ABB RAPID module: TargetDef.mod

MODULE TargetDef
CONST robtarget TOL0_0T1:=[[5.87495484961249, -209.948929822206, 55.199974607377],[0, 0.88684753706352, 0.462062166817809, 0],[-1, 0, -2, 0],[9E9,9E9,9E9,9E9,9E9,9E9]];
CONST robtarget TOL0_1T1:=[[5.62234055193414, -202.858739286579, 35.8261071491754],[0, 0.88684753706352, 0.462062166817809, 0],[-1, 0, -2, 0],[9E9,9E9,9E9,9E9,9E9,9E9]];
CONST robtarget TOL0_1T2:=[[4.98397898868433, -184.941680926626, 25.6156776604893],[0, 0.88684753706352, 0.462062166817809, 0],[-1, 0, -2, 0],[9E9,9E9,9E9,9E9,9E9,9E9]];
CONST robtarget TOL0_2T1:=[[4.89568379013019, -182.463476854714, 25.3040810063602],[0, 0.88684753706352, 0.462062166817809, 0],[-1, 0, -2, 0],[9E9,9E9,9E9,9E9,9E9,9E9]];
CONST robtarget TOL0_2T2:=[[4.80677150236914, -179.967952781144, 25.199974607377],[0, 0.88684753706352, 0.462062166817809, 0],[-1, 0, -2, 0],[9E9,9E9,9E9,9E9,9E9,9E9]];
CONST robtarget TOL0_3T1:=[[4.74728249481166, -178.298524485788, 25.1999746073769],[0, 0.88684753706352, 0.462062166817809, 0],[-1, 0, -2, 0],[9E9,9E9,9E9,9E9,9E9,9E9]];
CONST robtarget TOL0_4T1:=[[4.68786399989119, -176.629093681283, 25.199974607377],[0, 0.88684753706352, 0.462062166817809, 0],[-1, 0, -2, 0],[9E9,9E9,9E9,9E9,9E9,9E9]];
CONST robtarget TOL0_5T1:=[[4.11392451424888, -159.986640927652, 25.199974607377],[0, 0.88684753706352, 0.462062166817809, 0],[-1, 0, -2, 0],[9E9,9E9,9E9,9E9,9E9,9E9]];
CONST robtarget TOL0_6T1:=[[4.16406846873616, -158.042748709129, 25.1999105550075],[0, 0.88684753706352, 0.462062166817809, 0],[-1, 0, -2, 0],[9E9,9E9,9E9,9E9,9E9,9E9]];
CONST robtarget TOL0_7T1:=[[4.21439940943662, -156.098861429512, 25.1997536242781],[0, 0.88684753706352, 0.462062166817809, 0],[-1, 0, -2, 0],[9E9,9E9,9E9,9E9,9E9,9E9]];
CONST robtarget TOL0_8T1:=[[4.26487731018307, -154.154977990189, 25.199556654764],[0, 0.88684753706352, 0.462062166817809, 0],[-1, 1, -2, 0],[9E9,9E9,9E9,9E9,9E9,9E9]];
CONST robtarget TOL0_9T1:=[[4.31546214481006, -152.211097292488, 25.1993724860406],[0, 0.88684753706352, 0.462062166817809, 0],[-1, 1, -2, 0],[9E9,9E9,9E9,9E9,9E9,9E9]];
CONST robtarget TOL0_10T1:=[[4.36611388715329, -150.267218237672, 25.199253957683],[0, 0.88684753706352, 0.462062166817809, 0],[-1, 1, -2, 0],[9E9,9E9,9E9,9E9,9E9,9E9]];
CONST robtarget TOL0_11T1:=[[4.41679251104966, -148.32333972694, 25.1992539092665],[0, 0.88684753706352, 0.462062166817809, 0],[-1, 1, -2, 0],[9E9,9E9,9E9,9E9,9E9,9E9]];
CONST robtarget TOL0_12T1:=[[4.46745799033829, -146.379460661428, 25.1994251803665],[0, 0.88684753706352, 0.462062166817809, 0],[-1, 1, -2, 0],[9E9,9E9,9E9,9E9,9E9,9E9]];
CONST robtarget TOL0_13T1:=[[4.51807029885896, -144.435579942209, 25.1998206105581],[0, 0.88684753706352, 0.462062166817809, 0],[-1, 1, -2, 0],[9E9,9E9,9E9,9E9,9E9,9E9]];
CONST robtarget TOL0_14T1:=[[4.56860145931284, -142.491696832888, 25.2004340400337],[5.78808521166299E-05, -0.886847503502857, -0.462062165385235, -0.000239791711974077],[-1, 1, -2, 0],[9E9,9E9,9E9,9E9,9E9,9E9]];
CONST robtarget TOL0_15T1:=[[4.61907572015895, -140.547812172846, 25.2011438240197],[5.69174071655991E-06, 0.886847487536317, 0.462062177876197, 0.000278557770932622],[-1, 1, -2, 0],[9E9,9E9,9E9,9E9,9E9,9E9]];
CONST robtarget TOL0_16T1:=[[4.66953139612423, -138.603927209032, 25.2017324708743],[9.1999702878942E-05, 0.886847479230205, 0.462062185016766, 0.0002780226918304],[-1, 1, -2, 0],[9E9,9E9,9E9,9E9,9E9,9E9]];
CONST robtarget TOL0_17T1:=[[4.72000680111523, -136.660043190099, 25.2019991082225],[0.000194257642923755, 0.88684748453669, 0.462062172983582, 0.000223008078127303],[-1, 1, -2, 0],[9E9,9E9,9E9,9E9,9E9,9E9]];
CONST robtarget TOL0_18T1:=[[4.77054024868323, -134.716161363558, 25.2017428446979],[0.000305354655708716, 0.886847499341696, 0.462062127896507, 9.8151247610371E-05],[-1, 1, -2, 0],[9E9,9E9,9E9,9E9,9E9,9E9]];
CONST robtarget TOL0_19T1:=[[4.82117005178463, -132.772282975693, 25.2007627603113],[0.00041784330050476, 0.88684749715859, 0.462062040928341, -0.000111909145824577],[-1, 1, -2, 0],[9E9,9E9,9E9,9E9,9E9,9E9]];
CONST robtarget TOL0_20T1:=[[4.87193452255457, -130.828409271538, 25.1988578965212],[0.000523950911211992, 0.886847413047882, 0.462061914798928, -0.000422300923804722],[-1, 1, -2, 0],[9E9,9E9,9E9,9E9,9E9,9E9]];
CONST robtarget TOL0_21T1:=[[4.92287197203422, -128.884541494919, 25.1958272463483],[0.000615615291625375, 0.886847124286926, 0.46206177147994, -0.000847642992470561],[-1, 1, -2, 0],[9E9,9E9,9E9,9E9,9E9,9E9]];
CONST robtarget TOL0_22T1:=[[4.97401555483918, -126.940680952348, 25.1914949656618],[0.000644077831250294, 0.88684637798251, 0.46206172300607, -0.00143218564139338],[-1, 1, -2, 0],[9E9,9E9,9E9,9E9,9E9,9E9]];
CONST robtarget TOL0_23T1:=[[5.02537610710971, -124.996829121411, 25.1858015434017],[0.000673094305604695, 0.886844839539391, 0.462061777689024, -0.00216590056703986],[-1, 1, -2, 0],[9E9,9E9,9E9,9E9,9E9,9E9]];
CONST robtarget TOL0_24T1:=[[5.076958425822, -123.052987547218, 25.1787027683325],[0.000634581591898641, 0.886842136683072, 0.462062165434973, -0.00302938659633397],[-1, 1, -2, 0],[9E9,9E9,9E9,9E9,9E9,9E9]];
CONST robtarget TOL0_25T1:=[[5.12876731366958, -121.109157762365, 25.170161326942],[0.000531980538052365, 0.886837822825442, 0.462063048412129, -0.00401650283548481],[-1, 1, -2, 0],[9E9,9E9,9E9,9E9,9E9,9E9]];
CONST robtarget TOL0_26T1:=[[5.18080757241205, -119.165341299386, 25.1601399052154],[0.000368612428769883, 0.886831406094208, 0.462064598841902, -0.00512130714948808],[-1, 1, -2, 0],[9E9,9E9,9E9,9E9,9E9,9E9]];
CONST robtarget TOL0_27T1:=[[5.23308400297003, -117.221539690753, 25.1486011886477],[0.000147683364606522, 0.886822360123474, 0.462066996155013, -0.00633804693409372],[-1, 1, -2, 0],[9E9,9E9,9E9,9E9,9E9,9E9]];
CONST robtarget TOL0_28T1:=[[5.28560140550417, -115.277754468888, 25.1355078617056],[0.00012771642930868, -0.886810133767952, -0.462070424447913, 0.00766114779298364],[-1, 1, -2, 0],[9E9,9E9,9E9,9E9,9E9,9E9]];
CONST robtarget TOL0_29T1:=[[5.33836457940834, -113.3339871662, 25.1208226029927],[0.000454651248535902, -0.886794159972504, -0.462075070302794, 0.00908518219806045],[-1, 1, -2, 0],[9E9,9E9,9E9,9E9,9E9,9E9]];
CONST robtarget TOL0_30T1:=[[5.39137403539576, -111.390239241959, 25.1045122999512],[0.000830249094422553, -0.886773863455627, -0.462081120469981, 0.0106048990390756],[-1, 1, -2, 0],[9E9,9E9,9E9,9E9,9E9,9E9]];
CONST robtarget TOL0_31T1:=[[5.44461167530778, -109.446511823294, 25.0865606840709],[0.00125172016397042, -0.886748668292076, -0.462088759922859, 0.0122151721975377],[-1, 1, -2, 0],[9E9,9E9,9E9,9E9,9E9,9E9]];
CONST robtarget TOL0_32T1:=[[5.49805438484623, -107.502805944353, 25.0669557018495],[0.00171636213020819, -0.88671800451786, -0.462098170119577, 0.0139109933880112],[-1, 1, -2, 0],[9E9,9E9,9E9,9E9,9E9,9E9]];
CONST robtarget TOL0_33T1:=[[5.5516790497652, -105.559122639288, 25.0456852980213],[0.00222155399052518, -0.88668131405112, -0.462109527403577, 0.0156874693080021],[-1, 1, -2, 0],[9E9,9E9,9E9,9E9,9E9,9E9]];
CONST robtarget TOL0_34T1:=[[5.60546255581983, -103.615462942265, 25.0227374157007],[0.00276475085799574, -0.886638056102518, -0.462123001539547, 0.0175398138964316],[-1, 1, -2, 0],[9E9,9E9,9E9,9E9,9E9,9E9]];
CONST robtarget TOL0_35T1:=[[5.65938178871409, -101.671827887463, 24.9980999965197],[0.00334347917684389, -0.886587712061935, -0.462138754385235, 0.0194633415178935],[-1, 1, -2, 0],[9E9,9E9,9E9,9E9,9E9,9E9]];
CONST robtarget TOL0_36T1:=[[5.71341363405236, -99.7282185090801, 24.9717609807619],[0.0039553323360096, -0.886529789897628, -0.462156938690893, 0.0214534610270855],[-1, 1, -2, 0],[9E9,9E9,9E9,9E9,9E9,9E9]];
CONST robtarget TOL0_37T1:=[[5.76753497738014, -97.7846358413115, 24.9437083094337],[0.0045979493814297, -0.886463827969139, -0.46217769698422, 0.0235056796147047],[-1, 1, -2, 0],[9E9,9E9,9E9,9E9,9E9,9E9]];
CONST robtarget TOL0_38T1:=[[5.82172119826316, -95.8410808542579, 24.9139307673251],[0.00526886801727961, -0.886389397616001, -0.462201160277871, 0.0256156643784414],[-1, 1, -2, 0],[9E9,9E9,9E9,9E9,9E9,9E9]];
CONST robtarget TOL0_39T1:=[[5.87594113313077, -93.8975542480642, 24.8824204552068],[0.0059658038800925, -0.886306109324248, -0.46222744753722, 0.0277790658915003],[-1, 1, -2, 0],[9E9,9E9,9E9,9E9,9E9,9E9]];
CONST robtarget TOL0_40T1:=[[5.93016185341133, -91.9540566517558, 24.8491703063232],[0.00668656550503767, -0.886213614964218, -0.462256664707816, 0.0299915725997466],[-1, 1, -2, 0],[9E9,9E9,9E9,9E9,9E9,9E9]];
CONST robtarget TOL0_41T1:=[[5.98435043019924, -90.0105886943894, 24.8141732528904],[0.00742900624154073, -0.886111609894809, -0.462288903935541, 0.0322489375634248],[-1, 1, -2, 0],[9E9,9E9,9E9,9E9,9E9,9E9]];
CONST robtarget TOL0_42T1:=[[6.03847393420563, -88.0671510050547, 24.7774222262555],[0.00819102143652073, -0.885999835193581, -0.462324242939227, 0.0345469766469368],[-1, 1, -2, 0],[9E9,9E9,9E9,9E9,9E9,9E9]];
CONST robtarget TOL0_43T1:=[[6.09249943571575, -86.1237442128753, 24.7389101570525],[0.00897054595159374, -0.885878079539174, -0.462362744481674, 0.036881567383844],[-1, 1, -2, 0],[9E9,9E9,9E9,9E9,9E9,9E9]];
CONST robtarget TOL0_44T1:=[[6.14639400455496, -84.1803689470091, 24.6986299753559],[0.00976555199443826, -0.885746180751911, -0.462404455938409, 0.0392486484601787],[-1, 1, -2, 0],[9E9,9E9,9E9,9E9,9E9,9E9]];
CONST robtarget TOL0_45T1:=[[6.2001247100614, -82.2370258366481, 24.656574610829],[0.0105740472453268, -0.885604026997849, -0.462449408963551, 0.0416442197586716],[-1, 1, -2, 0],[9E9,9E9,9E9,9E9,9E9,9E9]];
CONST robtarget TOL0_46T1:=[[6.2536573860541, -80.2937157169943, 24.6127341371022],[0.0113941391592412, -0.885451558975314, -0.462497619103059, 0.0440643010271058],[-1, 1, -2, 0],[9E9,9E9,9E9,9E9,9E9,9E9]];
CONST robtarget TOL0_47T1:=[[6.30695259345345, -78.3504402383671, 24.5670871945443],[0.0122245639579626, -0.885288779804087, -0.462549084720571, 0.0465046300188573],[-1, 1, -2, 0],[9E9,9E9,9E9,9E9,9E9,9E9]];
CONST robtarget TOL0_48T1:=[[6.35996949801029, -76.4072012510752, 24.5196096457906],[0.0130635804060093, -0.885115740486263, -0.462603787181224, 0.0489612591343337],[-1, 1, -2, 0],[9E9,9E9,9E9,9E9,9E9,9E9]];
CONST robtarget TOL0_49T1:=[[6.41266726646654, -74.4640006050592, 24.4702773733228],[0.0139093019982725, -0.884932542700248, -0.462661691416617, 0.0514303945494261],[-1, 1, -2, 0],[9E9,9E9,9E9,9E9,9E9,9E9]];
CONST robtarget TOL0_50T1:=[[6.46500506498899, -72.520840150277, 24.4190662601734],[0.0147598699942932, -0.884739340551065, -0.462722746086731, 0.0539083089418833],[-1, 1, -2, 0],[9E9,9E9,9E9,9E9,9E9,9E9]];
CONST robtarget TOL0_51T1:=[[6.51694205924105, -70.5777217367015, 24.3659521900665],[0.0156134533099272, -0.884536339837173, -0.462786883826999, 0.0563913445565212],[-1, 1, -2, 0],[9E9,9E9,9E9,9E9,9E9,9E9]];
CONST robtarget TOL0_52T1:=[[6.56843741446033, -68.634647214319, 24.3109110475456],[0.0164682485958798, -0.884323797009536, -0.462854021586783, 0.0588759163984978],[-1, 1, -2, 0],[9E9,9E9,9E9,9E9,9E9,9E9]];
CONST robtarget TOL0_53T1:=[[6.61945029554181, -66.6916184331267, 24.25391871809],[0.0173224804765711, -0.884102017837447, -0.462924061054783, 0.0613585154843354],[-1, 1, -2, 0],[9E9,9E9,9E9,9E9,9E9,9E9]];
CONST robtarget TOL0_54T1:=[[6.66994435104448, -64.7486365163287, 24.1949689968205],[0.0181744089212188, -0.883871354009737, -0.462996889732181, 0.063835730744511],[-1, 1, -2, 0],[9E9,9E9,9E9,9E9,9E9,9E9]];
CONST robtarget TOL0_55T1:=[[6.7199019031716, -62.805699700113, 24.1341272804838],[0.0190218342643242, -0.883632185515794, -0.463072384977798, 0.066304576107361],[-1, 1, -2, 0],[9E9,9E9,9E9,9E9,9E9,9E9]];
CONST robtarget TOL0_56T1:=[[6.76931020604997, -60.8628054877942, 24.0714774096135],[0.0198573737794578, -0.883384829109368, -0.463150429844447, 0.0687648728705193],[-1, 0, -2, 0],[9E9,9E9,9E9,9E9,9E9,9E9]];
CONST robtarget TOL0_57T1:=[[6.81815645803619, -58.9199513943938, 24.0071027577105],[0.0206778301201626, -0.883129717086152, -0.46323088464036, 0.0712143079455536],[-1, 0, -2, 0],[9E9,9E9,9E9,9E9,9E9,9E9]];
CONST robtarget TOL0_58T1:=[[6.86642783302506, -56.9771349397499, 23.9410865196908],[0.0214816257464342, -0.882867352992543, -0.463313591712299, 0.0736497964008017],[-1, 0, -2, 0],[9E9,9E9,9E9,9E9,9E9,9E9]];
CONST robtarget TOL0_59T1:=[[6.91411150360364, -55.0343536436539, 23.8735118903307],[0.0222672059395263, -0.882598279750095, -0.46339838054372, 0.0760683181835714],[-1, 0, -2, 0],[9E9,9E9,9E9,9E9,9E9,9E9]];
CONST robtarget TOL0_60T1:=[[6.96119441598756, -53.0916050709859, 23.8044606758834],[0.023045541467769, -0.882323362092062, -0.463485011503932, 0.0784603838648393],[-1, 0, -2, 0],[9E9,9E9,9E9,9E9,9E9,9E9]];
CONST robtarget TOL0_61T1:=[[7.00766329729066, -51.1488868294857, 23.7340135480734],[0.0238379753498431, -0.882043756945659, -0.463573176999837, 0.0808113316972624],[-1, 0, -2, 0],[9E9,9E9,9E9,9E9,9E9,9E9]];
CONST robtarget TOL0_62T1:=[[7.05348992599602, -49.2062003980425, 23.6621651291686],[0.0246434226405345, -0.881760150918272, -0.463662654617083, 0.0831184737984602],[-1, 0, -2, 0],[9E9,9E9,9E9,9E9,9E9,9E9]];
CONST robtarget TOL0_63T1:=[[7.09858462534561, -47.2635630423646, 23.5885558995094],[0.0254603521153771, -0.881473231922942, -0.463753217597252, 0.0853795352627361],[-1, 0, -2, 0],[9E9,9E9,9E9,9E9,9E9,9E9]];
CONST robtarget TOL0_64T1:=[[7.14284253298126, -45.3209959322502, 23.5127389692874],[0.0262767684505692, -0.881183417162999, -0.46384470052432, 0.0875980054124462],[-1, 0, -2, 0],[9E9,9E9,9E9,9E9,9E9,9E9]];
CONST robtarget TOL0_65T1:=[[7.18616220901009, -43.3785195720567, 23.4342856300351],[0.0269162483623758, -0.880886836321344, -0.463937962561879, 0.0898635858610179],[-1, 0, -2, 0],[9E9,9E9,9E9,9E9,9E9,9E9]];
CONST robtarget TOL0_66T1:=[[7.22844016516217, -41.4361548561847, 23.3527545172302],[0.0273156512506206, -0.880582353172387, -0.464033139854085, 0.0922053121858804],[-1, 0, -2, 0],[9E9,9E9,9E9,9E9,9E9,9E9]];
CONST robtarget TOL0_67T1:=[[7.26957169093038, -39.493922882487, 23.2676974031319],[0.0274736194950504, -0.880270370217772, -0.464129743785235, 0.0946195354161044],[-1, 0, -2, 0],[9E9,9E9,9E9,9E9,9E9,9E9]];
CONST robtarget TOL0_68T1:=[[7.30945207826227, -37.5518447104956, 23.1786661163437],[0.0273882713081452, -0.879951240672993, -0.464227015451949, 0.0971029080789399],[-1, 0, -2, 0],[9E9,9E9,9E9,9E9,9E9,9E9]];
CONST robtarget TOL0_69T1:=[[7.34797711476068, -35.6099412503439, 23.0852149483144],[0.0270353507422883, -0.87962460427133, -0.464323980346725, 0.0996638683060276],[-1, 0, -2, 0],[9E9,9E9,9E9,9E9,9E9,9E9]];
CONST robtarget TOL0_70T1:=[[7.43410920658374, -35.2152949167019, 23.049134476302],[0.027387152036867, -0.879402536820145, -0.464393137984042, 0.101193554789508],[-1, 0, -2, 0],[9E9,9E9,9E9,9E9,9E9,9E9]];
CONST robtarget TOL0_71T1:=[[7.83197636578603, -33.6097358151834, 22.8847547435323],[0.0287458481344975, -0.878443440770914, -0.464690940547519, 0.107578470683722],[-1, 0, -2, 0],[9E9,9E9,9E9,9E9,9E9,9E9]];
CONST robtarget TOL0_72T1:=[[8.22945422240645, -32.0052187325015, 22.7096518119473],[0.0299679675605213, -0.877402453198319, -0.465012407313013, 0.114150414308576],[-1, 0, -2, 0],[9E9,9E9,9E9,9E9,9E9,9E9]];
CONST robtarget TOL0_73T1:=[[8.62647919807819, -30.4019739957621, 22.522482668734],[0.0310535472491881, -0.876276641963512, -0.465357816872208, 0.120900894241218],[-1, 0, -2, 0],[9E9,9E9,9E9,9E9,9E9,9E9]];
CONST robtarget TOL0_74T1:=[[9.02298779202067, -28.8002318707254, 22.3219045770051],[0.0320062367781418, -0.875061742490296, -0.465727744933963, 0.127828851343795],[-1, 0, -2, 0],[9E9,9E9,9E9,9E9,9E9,9E9]];
CONST robtarget TOL0_75T1:=[[9.41891881577311, -27.2002263124348, 22.106689574242],[0.0328307845960863, -0.873754414135797, -0.466122396477093, 0.134926924160703],[-1, 0, -2, 0],[9E9,9E9,9E9,9E9,9E9,9E9]];
CONST robtarget TOL0_76T1:=[[9.81421180453196, -25.6022037193409, 21.8760718212889],[0.0335410415525868, -0.872351878470698, -0.46654187882036, 0.142182537489597],[-1, 0, -2, 0],[9E9,9E9,9E9,9E9,9E9,9E9]];
CONST robtarget TOL0_77T1:=[[10.2088046734556, -24.0064128875366, 21.6294029478869],[0.0341394073310869, -0.870851111778797, -0.466986180215052, 0.149588600731706],[-1, 0, -2, 0],[9E9,9E9,9E9,9E9,9E9,9E9]];
CONST robtarget TOL0_78T1:=[[10.6026353833184, -22.4131025747239, 21.3660347119904],[0.0346270923135725, -0.869249101594861, -0.467455194957132, 0.15713880667112],[-1, 0, -2, 0],[9E9,9E9,9E9,9E9,9E9,9E9]];
CONST robtarget TOL0_79T1:=[[10.9956381087109, -20.8225410290283, 21.0852936408323],[0.0350053180038412, -0.86754286815456, -0.467948737621279, 0.16482711726006],[-1, 0, -2, 0],[9E9,9E9,9E9,9E9,9E9,9E9]];
CONST robtarget TOL0_80T1:=[[11.387735033502, -19.2350755024655, 20.7864043718172],[0.035275549555721, -0.865729392921139, -0.468466575321836, 0.172647970281056],[-1, 0, -2, 0],[9E9,9E9,9E9,9E9,9E9,9E9]];
CONST robtarget TOL0_81T1:=[[11.7788461517508, -17.6510732111494, 20.4685658049336],[0.0354395435717827, -0.863805699488511, -0.469008415288741, 0.180595843448654],[-1, 0, -2, 0],[9E9,9E9,9E9,9E9,9E9,9E9]];
CONST robtarget TOL0_82T1:=[[12.1688914672051, -16.0709013399982, 20.1309767973821],[0.035499089128212, -0.861768975535691, -0.469573873144648, 0.188664848700458],[-1, 0, -1, 0],[9E9,9E9,9E9,9E9,9E9,9E9]];
CONST robtarget TOL0_83T1:=[[12.5577737734797, -14.4949397020433, 19.7728616566787],[0.0354496734894093, -0.859619255222402, -0.470161502354852, 0.196840591351999],[-1, 0, -1, 0],[9E9,9E9,9E9,9E9,9E9,9E9]];
CONST robtarget TOL0_84T1:=[[12.9453200975713, -12.9236163390144, 19.3935496981315],[0.0352839590064922, -0.857358264143806, -0.470769168972642, 0.205105433097117],[-1, 0, -1, 0],[9E9,9E9,9E9,9E9,9E9,9E9]];
CONST robtarget TOL0_85T1:=[[13.3313368681544, -11.3573707185873, 18.9923973991323],[0.0350023271936787, -0.854984460453189, -0.471395831043085, 0.21345346085223],[-1, 0, -1, 0],[9E9,9E9,9E9,9E9,9E9,9E9]];
CONST robtarget TOL0_86T1:=[[13.715630356576, -9.79664234621814, 18.5687608492739],[0.0346091194395503, -0.852496634607658, -0.472040505657559, 0.221877123320074],[-1, 0, -1, 0],[9E9,9E9,9E9,9E9,9E9,9E9]];
CONST robtarget TOL0_87T1:=[[14.0980062151705, -8.24188693555804, 18.1219996102562],[0.0341140537110323, -0.849894694300878, -0.472702239067701, 0.2303645656758],[-1, 0, -1, 0],[9E9,9E9,9E9,9E9,9E9,9E9]];
CONST robtarget TOL0_88T1:=[[14.4782703339407, -6.6936249152833, 17.6514899462765],[0.0335188844077826, -0.847178241537506, -0.473379814829405, 0.238908062579636],[-1, 0, -1, 0],[9E9,9E9,9E9,9E9,9E9,9E9]];
CONST robtarget TOL0_89T1:=[[14.856319392745, -5.15244264550846, 17.1565742612497],[0.0328272708903672, -0.844345818016324, -0.474072416101428, 0.247503240738359],[-1, 0, -1, 0],[9E9,9E9,9E9,9E9,9E9,9E9]];
CONST robtarget TOL0_90T1:=[[15.2324495482948, -3.61913923974505, 16.6364277633281],[0.0320431726758495, -0.841395948739511, -0.474779283629122, 0.256145904449442],[-1, 0, -1, 0],[9E9,9E9,9E9,9E9,9E9,9E9]];
CONST robtarget TOL0_91T1:=[[15.6067133899127, -2.09441147356056, 16.0903883343992],[0.0311744453603097, -0.838325138427612, -0.475500514305436, 0.264836510194628],[-1, 0, -1, 0],[9E9,9E9,9E9,9E9,9E9,9E9]];
CONST robtarget TOL0_92T1:=[[15.9776026533308, -0.578260587893794, 15.5186930171285],[0.0302074534032609, -0.835141339137625, -0.476231675882653, 0.273550441981555],[-1, 0, -1, 0],[9E9,9E9,9E9,9E9,9E9,9E9]];
CONST robtarget TOL0_93T1:=[[16.3460386010615, 0.928181059726583, 14.9203842450379],[0.0291600686936652, -0.831836088634164, -0.476974944471034, 0.282300043192435],[-1, 0, -1, 0],[9E9,9E9,9E9,9E9,9E9,9E9]];
CONST robtarget TOL0_94T1:=[[16.7116757500925, 2.42427889302336, 14.2949178617212],[0.0280320714161996, -0.82841040669241, -0.477728767810928, 0.291076665951922],[-1, 0, -1, 0],[9E9,9E9,9E9,9E9,9E9,9E9]];
CONST robtarget TOL0_95T1:=[[17.0151361682334, 3.93476049963918, 13.6717584136658],[0.0260567021781286, -0.825274850857875, -0.478314666391687, 0.299094548141088],[-1, 0, -1, 0],[9E9,9E9,9E9,9E9,9E9,9E9]];
CONST robtarget TOL0_96T1:=[[17.1885483413104, 5.48153915463342, 13.0889076997537],[0.0218239495227135, -0.822800320403308, -0.478477261399255, 0.305913154825538],[-1, 0, -1, 0],[9E9,9E9,9E9,9E9,9E9,9E9]];
CONST robtarget TOL0_97T1:=[[17.2254385337467, 7.05325549652198, 12.5497391180146],[0.0144872412219819, -0.821000352955872, -0.478058340683713, 0.311783199019517],[-1, 0, -1, 0],[9E9,9E9,9E9,9E9,9E9,9E9]];
CONST robtarget TOL0_98T1:=[[17.1252319861591, 8.63730799664661, 12.0573412841479],[0.00524659813226371, -0.820201874224259, -0.477043854613766, 0.315706381788983],[-1, 0, -1, 0],[9E9,9E9,9E9,9E9,9E9,9E9]];
CONST robtarget TOL0_99T1:=[[16.8838655266047, 10.2220927847176, 11.6171916385159],[0.00597316665179748, 0.820436524121733, 0.475359131296763, -0.317619154743517],[-1, 0, -1, 0],[9E9,9E9,9E9,9E9,9E9,9E9]];
CONST robtarget TOL0_100T1:=[[16.496459258559, 11.7913593023744, 11.2323677652838],[0.019225135650213, 0.821720532595913, 0.472929037796034, -0.317401773276139],[-1, 0, -1, 0],[9E9,9E9,9E9,9E9,9E9,9E9]];
CONST robtarget TOL0_101T1:=[[15.9620388422879, 13.3292864997246, 10.9035216337546],[0.0343858161198326, 0.823952858276942, 0.469729414294668, -0.315077102204235],[0, 0, -1, 0],[9E9,9E9,9E9,9E9,9E9,9E9]];
CONST robtarget TOL0_102T1:=[[15.2975665242909, 14.8265997654873, 10.6230056722904],[0.0513144276670698, 0.827031767548874, 0.465745710339988, -0.310590112975424],[0, 0, -1, 0],[9E9,9E9,9E9,9E9,9E9,9E9]];
CONST robtarget TOL0_103T1:=[[14.967367080232, 15.4539259643929, 10.5171328666547],[0.0590775300410213, 0.828573423219684, 0.463798553078389, -0.30800459402525],[0, 0, -1, 0],[9E9,9E9,9E9,9E9,9E9,9E9]];
CONST robtarget TOL0_104T1:=[[13.8242741167196, 17.2551838840315, 10.2499142060585],[0.0836930125687464, 0.833774679307542, 0.457206753692931, -0.297955110998864],[0, 0, -1, 0],[9E9,9E9,9E9,9E9,9E9,9E9]];
CONST robtarget TOL0_105T1:=[[12.4848081223101, 18.9224226369913, 10.0402609053551],[0.109534625655401, 0.839498617006178, 0.449720616805198, -0.284597267463337],[0, 0, -1, 0],[9E9,9E9,9E9,9E9,9E9,9E9]];
CONST robtarget TOL0_106T1:=[[10.9536580099233, 20.4227808614128, 9.88079634359366],[0.135438074203304, 0.845217264609808, 0.441778026830691, -0.268507874505003],[0, 0, -1, 0],[9E9,9E9,9E9,9E9,9E9,9E9]];
CONST robtarget TOL0_107T1:=[[9.25279902191795, 21.733940718676, 9.76141824500081],[0.160711130131284, 0.850682329933611, 0.433745809055314, -0.249752035662573],[0, 0, -1, 0],[9E9,9E9,9E9,9E9,9E9,9E9]];
CONST robtarget TOL0_108T1:=[[7.40886096224591, 22.8377253427806, 9.67235716029097],[0.184787474070288, 0.855676877550213, 0.426005724317412, -0.228450855768669],[0, 0, -1, 0],[9E9,9E9,9E9,9E9,9E9,9E9]];
CONST robtarget TOL0_109T1:=[[5.44903033150683, 23.7213019041005, 9.60859755233264],[0.20715683426475, 0.860015923003412, 0.418948401521263, -0.204794763265019],[0, 0, -2, 0],[9E9,9E9,9E9,9E9,9E9,9E9]];
CONST robtarget TOL0_110T1:=[[3.40063086296732, 24.3731686868072, 9.56625582451045],[0.227129911032962, 0.863476298086857, 0.412995568241102, -0.179597735981233],[0, 0, -2, 0],[9E9,9E9,9E9,9E9,9E9,9E9]];
CONST robtarget TOL0_111T1:=[[1.29099086049644, 24.7818685137185, 9.54151159931365],[0.244587840350064, 0.866034249185732, 0.408359653076031, -0.152983206038509],[0, 0, -2, 0],[9E9,9E9,9E9,9E9,9E9,9E9]];
CONST robtarget TOL0_112T1:=[[-0.852267278068496, 24.9384128294188, 9.53145844273632],[0.259577705187279, 0.86767136716036, 0.405165412304917, -0.124927187799793],[0, 0, -2, 0],[9E9,9E9,9E9,9E9,9E9,9E9]];
CONST robtarget TOL0_113T1:=[[-3.00023476448621, 24.844012774621, 9.53644373163792],[0.271889307282029, 0.868342688426414, 0.403531423738877, -0.0960185924566771],[0, 0, -2, 0],[9E9,9E9,9E9,9E9,9E9,9E9]];
CONST robtarget TOL0_114T1:=[[-5.12366624708858, 24.502525867907, 9.55754302843019],[0.28135861594483, 0.868077486512614, 0.403439060009092, -0.0671991927223259],[0, 1, -2, 0],[9E9,9E9,9E9,9E9,9E9,9E9]];
CONST robtarget TOL0_115T1:=[[-7.19333271253106, 23.9178635833248, 9.59591180590405],[0.288314290128393, 0.866942341188987, 0.404733532419318, -0.0384267471548012],[0, 1, -2, 0],[9E9,9E9,9E9,9E9,9E9,9E9]];
CONST robtarget TOL0_116T1:=[[-9.17986849060492, 23.0950990283751, 9.65350899172734],[0.293085784728034, 0.864964080104485, 0.407240030693865, -0.00966541876041895],[0, 1, -2, 0],[9E9,9E9,9E9,9E9,9E9,9E9]];
CONST robtarget TOL0_117T1:=[[-11.0533207749818, 22.0440582483403, 9.73539475274919],[0.295695307915798, 0.862263102822051, 0.410766595359259, 0.0183692821098943],[0, 1, -2, 0],[9E9,9E9,9E9,9E9,9E9,9E9]];
CONST robtarget TOL0_118T1:=[[-12.7872263020506, 20.7794803940538, 9.84738095575494],[0.2964167184953, 0.858955230763517, 0.415060996665293, 0.0453586770936465],[0, 1, -2, 0],[9E9,9E9,9E9,9E9,9E9,9E9]];
CONST robtarget TOL0_119T1:=[[-14.3702073274265, 19.3317230411206, 9.99434809074609],[0.295555093865856, 0.855144094965721, 0.419892824553204, 0.0711742876601827],[0, 1, -2, 0],[9E9,9E9,9E9,9E9,9E9,9E9]];
CONST robtarget TOL0_120T1:=[[-14.8501607304607, 18.8164149185304, 10.0523405697373],[0.294965135682195, 0.853808338616108, 0.421558451563138, 0.0793433145090054],[0, 1, -2, 0],[9E9,9E9,9E9,9E9,9E9,9E9]];
CONST robtarget TOL0_121T1:=[[-16.2076741090664, 17.091805662966, 10.2716810818974],[0.292265376866975, 0.849475896643786, 0.426882422621381, 0.103648674680103],[0, 1, -2, 0],[9E9,9E9,9E9,9E9,9E9,9E9]];
CONST robtarget TOL0_122T1:=[[-17.3579077901645, 15.2330082223245, 10.5535971346291],[0.288191314532163, 0.845270097479071, 0.432176877743502, 0.125249251015019],[0, 1, -2, 0],[9E9,9E9,9E9,9E9,9E9,9E9]];
CONST robtarget TOL0_123T1:=[[-18.2679853277614, 13.2576263755874, 10.9164700516849],[0.282757246693219, 0.841580157683036, 0.437231498642144, 0.143595940861194],[-1, 1, -2, 0],[9E9,9E9,9E9,9E9,9E9,9E9]];
CONST robtarget TOL0_124T1:=[[-18.9282987581193, 11.2022331861768, 11.3709652323788],[0.275865633923922, 0.838802145713515, 0.441892833132222, 0.158239806599144],[-1, 1, -2, 0],[9E9,9E9,9E9,9E9,9E9,9E9]];
CONST robtarget TOL0_125T1:=[[-19.3366998057772, 9.10642946980709, 11.9227671757553],[0.267431534272727, 0.837226195476365, 0.446064871239216, 0.168993499079251],[-1, 1, -2, 0],[9E9,9E9,9E9,9E9,9E9,9E9]];
CONST robtarget TOL0_126T1:=[[-19.4965991647885, 7.00248777750436, 12.5659733328788],[0.257354967513303, 0.837025344316078, 0.449706252013001, 0.175844478358571],[-1, 1, -2, 0],[9E9,9E9,9E9,9E9,9E9,9E9]];
CONST robtarget TOL0_127T1:=[[-19.410921819497, 4.92186687191422, 13.2933999260707],[0.245839935005472, 0.8382198120052, 0.452739413887211, 0.178821967978035],[-1, 1, -2, 0],[9E9,9E9,9E9,9E9,9E9,9E9]];
CONST robtarget TOL0_128T1:=[[-19.0875426396446, 2.89348719239379, 14.097068940899],[0.235289232001358, 0.840599152710681, 0.454569819926168, 0.177195712641664],[-1, 1, -2, 0],[9E9,9E9,9E9,9E9,9E9,9E9]];
CONST robtarget TOL0_129T1:=[[-18.6102716309398, 0.906360223588791, 14.9291384799526],[0.223990247526092, 0.843722572428624, 0.456019413741289, 0.173224952240367],[-1, 1, -2, 0],[9E9,9E9,9E9,9E9,9E9,9E9]];
CONST robtarget TOL0_130T1:=[[-18.1201101074537, -1.09543148925224, 15.7172539691776],[0.21282322284174, 0.84676945109027, 0.457299572124969, 0.169011460717484],[-1, 1, -2, 0],[9E9,9E9,9E9,9E9,9E9,9E9]];
CONST robtarget TOL0_131T1:=[[-17.6268326464086, -3.11441539133411, 16.4581743933638],[0.20183330684969, 0.849710254539164, 0.458425216266941, 0.16462721727502],[-1, 1, -2, 0],[9E9,9E9,9E9,9E9,9E9,9E9]];
CONST robtarget TOL0_132T1:=[[-17.1270050146111, -5.14744898116223, 17.1548989732062],[0.19101493583257, 0.852557577273439, 0.459401526056578, 0.160028464903621],[-1, 1, -2, 0],[9E9,9E9,9E9,9E9,9E9,9E9]];
CONST robtarget TOL0_133T1:=[[-16.6241928732059, -7.19455251544644, 17.806847571344],[0.180407967373584, 0.855290530421207, 0.46024159112668, 0.155269931658141],[-1, 1, -2, 0],[9E9,9E9,9E9,9E9,9E9,9E9]];
CONST robtarget TOL0_134T1:=[[-16.1183745316094, -9.25418664761038, 18.4157406825447],[0.170018618749308, 0.857913209728371, 0.460953206051751, 0.150335410608257],[-1, 1, -2, 0],[9E9,9E9,9E9,9E9,9E9,9E9]];
CONST robtarget TOL0_135T1:=[[-15.6088409760248, -11.3245573025151, 18.9837212306742],[0.159864590327202, 0.860422186707043, 0.461545945455, 0.145231930427976],[-1, 1, -2, 0],[9E9,9E9,9E9,9E9,9E9,9E9]];
CONST robtarget TOL0_136T1:=[[-15.0960787303775, -13.4045453337182, 19.5121722473094],[0.149975300978849, 0.862815177086043, 0.462027176845585, 0.139958090664247],[-1, 1, -2, 0],[9E9,9E9,9E9,9E9,9E9,9E9]];
CONST robtarget TOL0_137T1:=[[-14.5808088220936, -15.493214306599, 20.0023703822673],[0.140372435895946, 0.865088826427405, 0.462406934533967, 0.134524081583902],[-1, 1, -2, 0],[9E9,9E9,9E9,9E9,9E9,9E9]];
CONST robtarget TOL0_138T1:=[[-14.0633726764923, -17.5896421566149, 20.4559695966065],[0.131074018363047, 0.867238384223207, 0.462696844175012, 0.128952770542435],[-1, 1, -2, 0],[9E9,9E9,9E9,9E9,9E9,9E9]];
CONST robtarget TOL0_139T1:=[[-13.5440096366595, -19.6929081775059, 20.8747204007841],[0.122103216966882, 0.869257873169228, 0.462908531594784, 0.12327710945837],[-1, 1, -2, 0],[9E9,9E9,9E9,9E9,9E9,9E9]];
CONST robtarget TOL0_140T1:=[[-13.0229591655849, -21.802091701674, 21.2603737525102],[0.113473998074668, 0.871147612677842, 0.463051803724335, 0.117509641112072],[-1, 1, -2, 0],[9E9,9E9,9E9,9E9,9E9,9E9]];
CONST robtarget TOL0_141T1:=[[-12.5004429779489, -23.9163253349126, 21.6147044837566],[0.105197548023017, 0.872909258683923, 0.463135958174091, 0.111660137202116],[-1, 1, -2, 0],[9E9,9E9,9E9,9E9,9E9,9E9]];
CONST robtarget TOL0_142T1:=[[-11.9766094698917, -26.0349538826794, 21.9395828092331],[0.0972844348343415, 0.8745449114134, 0.463169841914148, 0.105738518058062],[-1, 1, -2, 0],[9E9,9E9,9E9,9E9,9E9,9E9]];
CONST robtarget TOL0_143T1:=[[-11.4515880913778, -28.1573751184934, 22.2369029041797],[0.0897456004067372, 0.876056983401301, 0.463161765321256, 0.0997550409049293],[-1, 1, -2, 0],[9E9,9E9,9E9,9E9,9E9,9E9]];
CONST robtarget TOL0_144T1:=[[-10.9255078273131, -30.2829870216002, 22.5085572693407],[0.082607647437601, 0.877448336990899, 0.463118159041064, 0.0937121297546124],[-1, 1, -2, 0],[9E9,9E9,9E9,9E9,9E9,9E9]];
CONST robtarget TOL0_145T1:=[[-10.3985120967546, -32.4112341142956, 22.7564308997224],[0.0758954079375276, 0.878722264999561, 0.463045449924471, 0.0876126666200781],[-1, 1, -2, 0],[9E9,9E9,9E9,9E9,9E9,9E9]];
CONST robtarget TOL0_146T1:=[[-9.87080945530687, -34.541748928324, 22.982378047848],[0.0696194118664351, 0.879882234751099, 0.462950823272812, 0.0814673289841337],[-1, 1, -2, 0],[9E9,9E9,9E9,9E9,9E9,9E9]];
CONST robtarget TOL0_147T1:=[[-9.34262646956631, -36.6742116255785, 23.1882443954673],[0.0637908035852248, 0.880931931901293, 0.462840695078937, 0.0752871550362639],[-1, 1, -2, 0],[9E9,9E9,9E9,9E9,9E9,9E9]];
CONST robtarget TOL0_148T1:=[[-8.81419041693772, -38.8083023186704, 23.3758796746047],[0.0583825925832353, 0.88187519634327, 0.46272291516522, 0.0691022050211185],[-1, 1, -2, 0],[9E9,9E9,9E9,9E9,9E9,9E9]];
CONST robtarget TOL0_149T1:=[[-8.28568435468992, -40.9437188492464, 23.5471407678994],[0.0533472635017263, 0.882715691629315, 0.462605067045612, 0.0629573599508624],[-1, 1, -2, 0],[9E9,9E9,9E9,9E9,9E9,9E9]];
CONST robtarget TOL0_150T1:=[[-7.75710200855048, -43.0802271939391, 23.7038999132041],[0.048685885410195, 0.883459810652129, 0.462489590612448, 0.0568491521437229],[-1, 1, -2, 0],[9E9,9E9,9E9,9E9,9E9,9E9]];
CONST robtarget TOL0_151T1:=[[-7.22838727942678, -45.2176096718404, 23.8480344906063],[0.0444078950852048, 0.884112374799878, 0.462378731687064, 0.0507853922233948],[-1, 1, -2, 0],[9E9,9E9,9E9,9E9,9E9,9E9]];
CONST robtarget TOL0_152T1:=[[-6.69948509040722, -47.3556484213305, 23.9814305011278],[0.0404447801603883, 0.884677513200354, 0.462277822658423, 0.0448233429543472],[-1, 1, -2, 0],[9E9,9E9,9E9,9E9,9E9,9E9]];
CONST robtarget TOL0_153T1:=[[-6.54114552962392, -47.943030101082, 24.0174859657964],[0.039374611646011, 0.884818340956773, 0.462253349183249, 0.0432201877957459],[-1, 1, -2, 0],[9E9,9E9,9E9,9E9,9E9,9E9]];
CONST robtarget TOL0_154T1:=[[-6.57084359592528, -49.7143900827433, 24.0663889829553],[0.03869304390063, 0.884878175767734, 0.462251536204324, 0.0426260446254812],[-1, 1, -2, 0],[9E9,9E9,9E9,9E9,9E9,9E9]];
CONST robtarget TOL0_155T1:=[[-6.60030974493776, -51.4857852378788, 24.1141438239073],[0.0379741305375769, 0.884939950752581, 0.46224974685858, 0.0420050056673457],[-1, 1, -2, 0],[9E9,9E9,9E9,9E9,9E9,9E9]];
CONST robtarget TOL0_156T1:=[[-6.62954325240327, -53.257214932897, 24.160743984258],[0.03721785808578, 0.885003508041735, 0.462247973262702, 0.0413573815401012],[-1, 1, -2, 0],[9E9,9E9,9E9,9E9,9E9,9E9]];
CONST robtarget TOL0_157T1:=[[-6.6585433828397, -55.0286785371064, 24.2061828638426],[0.0364251103255965, 0.88506868087446, 0.462246174321102, 0.0406831144139272],[-1, 1, -2, 0],[9E9,9E9,9E9,9E9,9E9,9E9]];
CONST robtarget TOL0_158T1:=[[-6.6873091707605, -56.8001754775931, 24.2504516594229],[0.0356164757158764, 0.88513534147139, 0.462243585037126, 0.0399720155600327],[-1, 1, -2, 0],[9E9,9E9,9E9,9E9,9E9,9E9]];
CONST robtarget TOL0_159T1:=[[-6.71583980311863, -58.5717051409716, 24.2935428788471],[0.0348009122070444, 0.885203318465326, 0.462239940250233, 0.0392201367283948],[-1, 1, -2, 0],[9E9,9E9,9E9,9E9,9E9,9E9]];
CONST robtarget TOL0_160T1:=[[-6.74413457315251, -60.3432668868342, 24.335450005417],[0.0339787181729264, 0.885272408822688, 0.46223531518711, 0.0384281444058096],[-1, 1, -2, 0],[9E9,9E9,9E9,9E9,9E9,9E9]];
CONST robtarget TOL0_161T1:=[[-6.77219277484988, -62.1148600748615, 24.3761665236126],[0.0331502211243416, 0.885342401638604, 0.462229787559614, 0.037596784341091],[-1, 1, -2, 0],[9E9,9E9,9E9,9E9,9E9,9E9]];
CONST robtarget TOL0_162T1:=[[-6.80001521916989, -63.8864839303779, 24.4156920434949],[0.0323155433289327, 0.885413077710598, 0.462223445482568, 0.0367270190000014],[-1, 1, -2, 0],[9E9,9E9,9E9,9E9,9E9,9E9]];
CONST robtarget TOL0_163T1:=[[-6.82760915391543, -65.6581371279869, 24.4540510196721],[0.0314705173280732, 0.885484199040336, 0.462216519541101, 0.0358221838015254],[-1, 1, -2, 0],[9E9,9E9,9E9,9E9,9E9,9E9]];
CONST robtarget TOL0_164T1:=[[-6.8549834753818, -67.4298182145868, 24.4912736728431],[0.0306138264791331, 0.885555530724849, 0.462209136496061, 0.0348842338385297],[-1, 1, -2, 0],[9E9,9E9,9E9,9E9,9E9,9E9]];
CONST robtarget TOL0_165T1:=[[-6.88214706060234, -69.2015257418041, 24.5273900296316],[0.0297459321372872, 0.885626838550497, 0.462201364736033, 0.0339143155095987],[-1, 1, -2, 0],[9E9,9E9,9E9,9E9,9E9,9E9]];
CONST robtarget TOL0_166T1:=[[-6.90910878641529, -70.9732582612964, 24.5624301179233],[0.0288673364953879, 0.885697885450896, 0.462193273656697, 0.032913680711508],[-1, 1, -2, 0],[9E9,9E9,9E9,9E9,9E9,9E9]];
CONST robtarget TOL0_167T1:=[[-6.93587752945251, -72.7450143247525, 24.5964239669314],[0.0279785846353445, 0.885768432711658, 0.462184933304451, 0.0318836923786601],[-1, 1, -2, 0],[9E9,9E9,9E9,9E9,9E9,9E9]];
CONST robtarget TOL0_168T1:=[[-6.96246216612661, -74.5167924838946, 24.629401607269],[0.0270802666639738, 0.885838241270577, 0.462176413991036, 0.0308258302474702],[-1, 1, -2, 0],[9E9,9E9,9E9,9E9,9E9,9E9]];
CONST robtarget TOL0_169T1:=[[-6.98887157262055, -76.2885912904786, 24.6613930710228],[0.0261730199358578, 0.885907073112755, 0.462167785879364, 0.0297416968512933],[-1, 1, -2, 0],[9E9,9E9,9E9,9E9,9E9,9E9]];
CONST robtarget TOL0_170T1:=[[-7.01511476686795, -78.0604094148144, 24.6924247368129],[0.0252575330175447, 0.885974692625851, 0.462159118562782, 0.028633026065519],[-1, 1, -2, 0],[9E9,9E9,9E9,9E9,9E9,9E9]];
CONST robtarget TOL0_171T1:=[[-7.04120148983964, -79.8322459992297, 24.7225083528119],[0.0243345523095351, 0.886040867889213, 0.462150480638381, 0.0275016952157162],[-1, 1, -2, 0],[9E9,9E9,9E9,9E9,9E9,9E9]];
CONST robtarget TOL0_172T1:=[[-7.06714170161695, -81.6041003036633, 24.7516520019587],[0.0234049313723166, 0.886105373003747, 0.462141937823974, 0.0263496949820964],[-1, 1, -2, 0],[9E9,9E9,9E9,9E9,9E9,9E9]];
CONST robtarget TOL0_173T1:=[[-7.09294535851427, -83.3759715890191, 24.7798637122967],[0.022470082543401, 0.88616799071574, 0.462133542112832, 0.0251788974255734],[-1, 1, -2, 0],[9E9,9E9,9E9,9E9,9E9,9E9]];
CONST robtarget TOL0_174T1:=[[-7.11862242030958, -85.1478591153642, 24.8071515596534],[0.0215310676654325, 0.886228512500455, 0.462125354031602, 0.0239915384580629],[-1, 1, -2, 0],[9E9,9E9,9E9,9E9,9E9,9E9]];
CONST robtarget TOL0_175T1:=[[-7.14418284780567, -86.9197621425125, 24.8335236387036],[0.0205888602110719, 0.886286740916632, 0.462117434658868, 0.0227900920334054],[-1, 1, -2, 0],[9E9,9E9,9E9,9E9,9E9,9E9]];
CONST robtarget TOL0_176T1:=[[-7.16963660159678, -88.691679930324, 24.85898804639],[0.0196444969518259, 0.886342491757068, 0.462109841315673, 0.021577201036868],[-1, 1, -2, 0],[9E9,9E9,9E9,9E9,9E9,9E9]];
CONST robtarget TOL0_177T1:=[[-7.19499364202744, -90.4636117387061, 24.8835528820602],[0.0186990811894058, 0.886395595963793, 0.462102626988536, 0.0203556859122318],[-1, 1, -2, 0],[9E9,9E9,9E9,9E9,9E9,9E9]];
CONST robtarget TOL0_178T1:=[[-7.22026415906436, -92.2355568453319, 24.9072262230203],[0.0177537868116957, 0.886445901532522, 0.462095839750076, 0.0191285544595607],[-1, 1, -2, 0],[9E9,9E9,9E9,9E9,9E9,9E9]];
CONST robtarget TOL0_179T1:=[[-7.24545934716298, -94.007514597632, 24.930016046348],[0.0168098635974773, 0.88649327538598, 0.462089522181154, 0.0178990131477915],[-1, 1, -2, 0],[9E9,9E9,9E9,9E9,9E9,9E9]];
CONST robtarget TOL0_180T1:=[[-7.27059067291594, -95.7794843602319, 24.9519303051068],[0.0158686383792753, 0.886537605440941, 0.462083710776268, 0.0166704736065185],[-1, 1, -2, 0],[9E9,9E9,9E9,9E9,9E9,9E9]];
CONST robtarget TOL0_181T1:=[[-7.29566960252566, -97.5514654978175, 24.9729769553915],[0.0149315181094865, 0.886578802501652, 0.462078435384309, 0.0154465618981082],[-1, 1, -2, 0],[9E9,9E9,9E9,9E9,9E9,9E9]];
CONST robtarget TOL0_182T1:=[[-7.3207076018852, -99.3234573751063, 24.9931639594113],[0.013999968090584, 0.886616802018349, 0.462073719069452, 0.0142311425241532],[-1, 1, -2, 0],[9E9,9E9,9E9,9E9,9E9,9E9]];
CONST robtarget TOL0_183T1:=[[-7.34571613690127, -101.095459356737, 25.0124992967216],[0.013075417536147, 0.886651565751382, 0.462069578891134, 0.0130283794175794],[-1, 1, -2, 0],[9E9,9E9,9E9,9E9,9E9,9E9]];
CONST robtarget TOL0_184T1:=[[-7.37070667236736, -102.867470807609, 25.030990936327],[0.0121595131909455, 0.886683083368959, 0.462066021604572, 0.0118426173120142],[-1, 1, -2, 0],[9E9,9E9,9E9,9E9,9E9,9E9]];
CONST robtarget TOL0_185T1:=[[-7.39569067250727, -104.63949109274, 25.0486468483312],[0.0112540229090199, 0.886711373584813, 0.462063045129794, 0.0106784478778441],[-1, 1, -2, 0],[9E9,9E9,9E9,9E9,9E9,9E9]];
CONST robtarget TOL0_186T1:=[[-7.42067981169834, -106.411519603206, 25.0654681478275],[0.0103608168906342, 0.886736485116131, 0.462060638660858, 0.00954073569326912],[-1, 1, -2, 0],[9E9,9E9,9E9,9E9,9E9,9E9]];
CONST robtarget TOL0_187T1:=[[-7.44568675794295, -108.183555831958, 25.0814285135408],[0.00948187404938943, 0.886758497314232, 0.462058782492553, 0.00843463259521849],[-1, 1, -2, 0],[9E9,9E9,9E9,9E9,9E9,9E9]];
CONST robtarget TOL0_188T1:=[[-7.47072446486959, -109.955599296986, 25.0964947676554],[0.00861928369429008, 0.886777520475811, 0.462057447982504, 0.00736558831769055],[-1, 1, -2, 0],[9E9,9E9,9E9,9E9,9E9,9E9]];
CONST robtarget TOL0_189T1:=[[-7.49580588511714, -111.72764951641, 25.1106337374164],[0.0077752501343488, 0.886793695558858, 0.46205659767654, 0.00633936479404148],[-1, 1, -2, 0],[9E9,9E9,9E9,9E9,9E9,9E9]];
CONST robtarget TOL0_190T1:=[[-7.52094397026718, -113.499706008499, 25.1238122554261],[0.00695209841453766, 0.886807193280896, 0.462056185621002, 0.00536205205720291],[-1, 1, -2, 0],[9E9,9E9,9E9,9E9,9E9,9E9]];
CONST robtarget TOL0_191T1:=[[-7.54615167079334, -115.271768291692, 25.1359971599557],[0.00615228023593474, 0.8868182125129, 0.462056157896262, 0.00444008484926977],[-1, 1, -2, 0],[9E9,9E9,9E9,9E9,9E9,9E9]];
CONST robtarget TOL0_192T1:=[[-7.57144193601533, -117.043835884628, 25.1471552938486],[0.00537839268800403, 0.886826977834939, 0.462056453328572, 0.00358025329604011],[-1, 1, -2, 0],[9E9,9E9,9E9,9E9,9E9,9E9]];
CONST robtarget TOL0_193T1:=[[-7.59682771409274, -118.815908306176, 25.1572535027561],[0.00463320282505451, 0.886833736114481, 0.462057004531966, 0.00278971033623931],[-1, 1, -2, 0],[9E9,9E9,9E9,9E9,9E9,9E9]];
CONST robtarget TOL0_194T1:=[[-7.62231922963412, -120.587985048012, 25.1662691832259],[0.0039195805998872, 0.886838752001448, 0.4620577398421, 0.00207602708195741],[-1, 1, -2, 0],[9E9,9E9,9E9,9E9,9E9,9E9]];
CONST robtarget TOL0_195T1:=[[-7.64791477467037, -122.360065507354, 25.174221907386],[0.00324053812772405, 0.886842302033931, 0.462058584883698, 0.00144719420806597],[-1, 1, -2, 0],[9E9,9E9,9E9,9E9,9E9,9E9]];
CONST robtarget TOL0_196T1:=[[-7.67360939862965, -124.132149061767, 25.181141798402],[0.0025992514690445, 0.886844667196804, 0.462059464851378, 0.000911645571989325],[-1, 1, -2, 0],[9E9,9E9,9E9,9E9,9E9,9E9]];
CONST robtarget TOL0_197T1:=[[-7.69939815257459, -125.904235089148, 25.1870589861849],[0.0019990696455256, 0.886846123799991, 0.462060307397114, 0.000478277710666103],[-1, 1, -2, 0],[9E9,9E9,9E9,9E9,9E9,9E9]];
CONST robtarget TOL0_198T1:=[[-7.72527608981545, -127.676322967766, 25.1920036077173],[0.00144352082039246, 0.88684693233044, 0.462061046163147, 0.000156468357065677],[-1, 1, -2, 0],[9E9,9E9,9E9,9E9,9E9,9E9]];
CONST robtarget TOL0_199T1:=[[-7.75123825884651, -129.448412093672, 25.1959961528978],[0.00101166433542418, 0.886847298511531, 0.462061504657849, -0.000107570429472382],[-1, 1, -2, 0],[9E9,9E9,9E9,9E9,9E9,9E9]];
CONST robtarget TOL0_200T1:=[[-7.77727973760562, -131.220501817879, 25.1990751714935],[0.000639976666744541, 0.886847435580532, 0.462061849918151, -0.000251563741665539],[-1, 1, -2, 0],[9E9,9E9,9E9,9E9,9E9,9E9]];
CONST robtarget TOL0_201T1:=[[-7.80339558291485, -132.992591520107, 25.2012673263357],[0.000337172875398902, 0.886847468844766, 0.462062057142553, -0.00032964719952443],[-1, 1, -2, 0],[9E9,9E9,9E9,9E9,9E9,9E9]];
CONST robtarget TOL0_202T1:=[[-7.82957987023434, -134.764680695173, 25.2026210292041],[9.97706163052248E-05, 0.886847465174978, 0.462062159482721, -0.000352608430609474],[-1, 1, -2, 0],[9E9,9E9,9E9,9E9,9E9,9E9]];
CONST robtarget TOL0_203T1:=[[-7.85582237226959, -136.536769333982, 25.2032591902318],[7.63601753318885E-05, -0.886847459217866, -0.462062190798779, 0.000331786336365523],[-1, 1, -2, 0],[9E9,9E9,9E9,9E9,9E9,9E9]];
CONST robtarget TOL0_204T1:=[[-7.88211169615124, -138.308857553145, 25.2033233629971],[0.000195889074552846, -0.886847463607737, -0.462062182076528, 0.000278952810838877],[-1, 1, -2, 0],[9E9,9E9,9E9,9E9,9E9,9E9]];
CONST robtarget TOL0_205T1:=[[-7.90843644954845, -140.080945469817, 25.2029551229297],[0.000263922178407408, -0.886847478045912, -0.462062158699036, 0.000206220937672317],[-1, 1, -2, 0],[9E9,9E9,9E9,9E9,9E9,9E9]];
CONST robtarget TOL0_206T1:=[[-7.9347852404278, -141.853033201824, 25.2022960619861],[0.000285906107501688, -0.886847496715285, -0.462062138631075, 0.000125980979006009],[-1, 1, -2, 0],[9E9,9E9,9E9,9E9,9E9,9E9]];
CONST robtarget TOL0_207T1:=[[-7.96114667597959, -143.625120863301, 25.2014666595926],[0, 0.88684753706352, 0.462062166817809, 0],[-1, 1, -2, 0],[9E9,9E9,9E9,9E9,9E9,9E9]];
CONST robtarget TOL0_208T1:=[[-7.98750936652624, -145.397208583346, 25.2006527033653],[0, 0.88684753706352, 0.462062166817809, 0],[-1, 1, -2, 0],[9E9,9E9,9E9,9E9,9E9,9E9]];
CONST robtarget TOL0_209T1:=[[-8.01386191884848, -147.169296478218, 25.1999767250408],[0, 0.88684753706352, 0.462062166817809, 0],[-1, 0, -2, 0],[9E9,9E9,9E9,9E9,9E9,9E9]];
CONST robtarget TOL0_210T1:=[[-8.04019530389439, -148.941384641741, 25.1995480711765],[0, 0.88684753706352, 0.462062166817809, 0],[-1, 0, -2, 0],[9E9,9E9,9E9,9E9,9E9,9E9]];
CONST robtarget TOL0_211T1:=[[-8.06651081840988, -150.713473050365, 25.1993466691209],[0, 0.88684753706352, 0.462062166817809, 0],[-1, 0, -2, 0],[9E9,9E9,9E9,9E9,9E9,9E9]];
CONST robtarget TOL0_212T1:=[[-8.09281255906433, -152.48556164795, 25.1993200914208],[0, 0.88684753706352, 0.462062166817809, 0],[-1, 0, -2, 0],[9E9,9E9,9E9,9E9,9E9,9E9]];
CONST robtarget TOL0_213T1:=[[-8.11910462252689, -154.257650378354, 25.1994159106226],[0, 0.88684753706352, 0.462062166817809, 0],[-1, 0, -2, 0],[9E9,9E9,9E9,9E9,9E9,9E9]];
CONST robtarget TOL0_214T1:=[[-8.14539110546667, -156.029739185438, 25.1995816992726],[0, 0.88684753706352, 0.462062166817809, 0],[-1, 0, -2, 0],[9E9,9E9,9E9,9E9,9E9,9E9]];
CONST robtarget TOL0_215T1:=[[-8.17167610455328, -157.801828013062, 25.1997650299172],[0, 0.88684753706352, 0.462062166817809, 0],[-1, 0, -2, 0],[9E9,9E9,9E9,9E9,9E9,9E9]];
CONST robtarget TOL0_216T1:=[[-8.19796371645577, -159.573916805089, 25.1999134751032],[0, 0.88684753706352, 0.462062166817809, 0],[-1, 0, -2, 0],[9E9,9E9,9E9,9E9,9E9,9E9]];
CONST robtarget TOL0_217T1:=[[-8.22425803784341, -161.346005505381, 25.199974607377],[0, 0.88684753706352, 0.462062166817809, 0],[-1, 0, -2, 0],[9E9,9E9,9E9,9E9,9E9,9E9]];
CONST robtarget TOL0_218T1:=[[-6.27565355284332, -177.026616849828, 25.199974607377],[0, 0.88684753706352, 0.462062166817809, 0],[-1, 0, -2, 0],[9E9,9E9,9E9,9E9,9E9,9E9]];
CONST robtarget TOL0_219T1:=[[-4.9045912867972, -177.710222759888, 25.199974607377],[0, 0.88684753706352, 0.462062166817809, 0],[-1, 0, -2, 0],[9E9,9E9,9E9,9E9,9E9,9E9]];
CONST robtarget TOL0_220T1:=[[-3.44531023421689, -178.177497756452, 25.1999746073771],[0, 0.88684753706352, 0.462062166817809, 0],[-1, 0, -2, 0],[9E9,9E9,9E9,9E9,9E9,9E9]];
CONST robtarget TOL0_221T1:=[[-1.93076759838084, -178.414930359914, 25.199974607377],[0, 0.88684753706352, 0.462062166817809, 0],[-1, 0, -2, 0],[9E9,9E9,9E9,9E9,9E9,9E9]];
CONST robtarget TOL0_222T1:=[[-0.399218636393755, -178.420811620707, 25.1999746073769],[0, 0.88684753706352, 0.462062166817809, 0],[-1, 0, -2, 0],[9E9,9E9,9E9,9E9,9E9,9E9]];
CONST robtarget TOL0_223T1:=[[1.11490597984312, -178.190406037047, 25.199974607377],[0, 0.88684753706352, 0.462062166817809, 0],[-1, 0, -2, 0],[9E9,9E9,9E9,9E9,9E9,9E9]];
CONST robtarget TOL0_224T1:=[[2.57813623007382, -177.73306670033, 25.199974607377],[0, 0.88684753706352, 0.462062166817809, 0],[-1, 0, -2, 0],[9E9,9E9,9E9,9E9,9E9,9E9]];
CONST robtarget TOL0_225T1:=[[3.95352770741732, -177.057599659804, 25.199974607377],[0, 0.88684753706352, 0.462062166817809, 0],[-1, 0, -2, 0],[9E9,9E9,9E9,9E9,9E9,9E9]];
CONST robtarget TOL0_226T1:=[[5.20773790579511, -176.177959456692, 25.199974607377],[0, 0.88684753706352, 0.462062166817809, 0],[-1, 0, -2, 0],[9E9,9E9,9E9,9E9,9E9,9E9]];
CONST robtarget TOL0_227T1:=[[7.16857129290258, -174.631777635337, 25.3040810063602],[0, 0.88684753706352, 0.462062166817809, 0],[-1, 0, -2, 0],[9E9,9E9,9E9,9E9,9E9,9E9]];
CONST robtarget TOL0_227T2:=[[9.11579565981418, -173.096326975422, 25.6156776604893],[0, 0.88684753706352, 0.462062166817809, 0],[-1, 0, -2, 0],[9E9,9E9,9E9,9E9,9E9,9E9]];
CONST robtarget TOL0_228T1:=[[23.1939472605264, -161.99523994456, 35.8261071491754],[0, 0.88684753706352, 0.462062166817809, 0],[-1, 1, -2, 0],[9E9,9E9,9E9,9E9,9E9,9E9]];
CONST robtarget TOL0_228T2:=[[28.7649944287146, -157.602285441643, 55.199974607377],[0, 0.88684753706352, 0.462062166817809, 0],[-1, 1, -2, 0],[9E9,9E9,9E9,9E9,9E9,9E9]];
ENDMODULE
